TYPE AlarmLimitsA :
STRUCT
	FireExtractTemperature: REAL := 45;
	FireExtractPressureTemperature: REAL := 38;
	FireExtractPressure: REAL := 170;
	Freeze: REAL := 8;
END_STRUCT
END_TYPE

(* stored: Version 1.1.0.1, ProductVersion 3.1.4024.6
   DUT AlarmLimitsA: Id {4247b6ac-ae38-485c-8b72-e24b66dd451c} *)
